TYPE ST_Alarmes :
STRUCT
	Id          : UINT;          // ID unique
    Libelle     : STRING(80);    // Texte affiché
    Active      : BOOL;          // Vrai si alarme à afficher
END_STRUCT
END_TYPE

(* stored: Version 1.1.0.1, ProductVersion 3.1.4024.15
   DUT ST_Alarmes: Id {643ab072-79da-4808-9822-896afe800bf5} *)
